// TIA Portal V18 export
TYPE "batchID_ShW"
// stored: IsFailsafeCompliant false
   STRUCT
      _1 : Struct
         "name" : String[48];
         code : String[48];
         number : DInt;
      END_STRUCT;
      _2 : Struct
         "name" : String[48];
         code : String[48];
         number : DInt;
      END_STRUCT;
      _3 : Struct
         "name" : String[48];
         code : String[48];
         number : DInt;
      END_STRUCT;
      _4 : Struct
         "name" : String[48];
         code : String[48];
         number : DInt;
      END_STRUCT;
      _5 : Struct
         "name" : String[48];
         code : String[48];
         number : DInt;
      END_STRUCT;
      _6 : Struct
         "name" : String[48];
         code : String[48];
         number : DInt;
      END_STRUCT;
      _7 : Struct
         "name" : String[48];
         code : String[48];
         number : DInt;
      END_STRUCT;
      _8 : Struct
         "name" : String[48];
         code : String[48];
         number : DInt;
      END_STRUCT;
      _9 : Struct
         "name" : String[48];
         code : String[48];
         number : DInt;
      END_STRUCT;
      _10 : Struct
         "name" : String[48];
         code : String[48];
         number : DInt;
      END_STRUCT;
   END_STRUCT;
END_TYPE
